FUNCTION_BLOCK Clearing IMPLEMENTS ITF_PackMLState
VAR
END_VAR

METHOD CyclicLogic : BOOL
VAR_INPUT
END_VAR
END_METHOD

{warning 'add method implementation '}
METHOD EStop : BOOL
END_METHOD

{warning 'add method implementation '}
METHOD Reset : BOOL
END_METHOD

{warning 'add method implementation '}
METHOD Start : BOOL
END_METHOD

{warning 'add method implementation '}
METHOD Stop : BOOL
END_METHOD

END_FUNCTION_BLOCK

(* stored: Version 1.1.0.1, ProductVersion 3.1.4024.12
   POU Clearing: Id {a6f0b167-4c13-4b94-937d-2718ad9d0c4c}, SpecialFunc None
   Method CyclicLogic: Id {a9ea858b-2722-4d90-afa7-e9b930e801d5}
   Method EStop: Id {549d8647-c1b6-4564-b600-4c8d59c32a93}
   Method Reset: Id {e79bc8a8-656b-4d44-a6fa-8bfcb2bf92df}
   Method Start: Id {d70cc64b-471d-4407-83ae-9ec920ed16af}
   Method Stop: Id {020009b6-cd1f-4ff7-99d7-2fbd1f97d684} *)
